// TIA Portal V20 export
DATA_BLOCK "MP101"   // DB181
// stored: MemoryReserve 100
   VAR
      "KISTLER 100KN PRESS POWER TRIPPED E202CB" : Bool;
      "KISTLER 100KN PRESS POWER TRIPPED E208CB" : Bool;
      "KISTLER 30KN PRESS POWER TRIPPED E214CB" : Bool;
      SPARE : Bool;
      SPARE_1 : Bool;
      "E8404PWS CONTROLLER POWER SMPS AC POWER TRIPPED E320CB" : Bool;
      "E8704PWS SAFETY POWER SMPS AC POWER TRIPPED E326CB" : Bool;
      "E8804PWS CONTRL POWER SMPS AC POWER TRIPPED E332CB" : Bool;
      "PROCESSOR POWER ON TIPPRED E4120CB" : Bool;
      "PROGRAMING POWER OUTLET TRPPED E4126CB" : Bool;
      SPARE_2 : Bool;
      "PANEL LED POWER TRIPPED E4304CB" : Bool;
      SPARE_3 : Bool;
      "PLC POWER SMPS DC OK E4404PWS" : Bool;
      "CONTROL LEVEL HUB POWER TRIPPED E4420CB" : Bool;
      "MAIN HMI POWER TRIPPED E4426CB" : Bool;
      "PORTABLE HMI POWER TIPPED E4432CB" : Bool;
      "PORTABLE HMI POWER TIPPED E4456CB" : Bool;
      "120VAC HEATER-1 POWER TR PRIMARY TRIPPED E5100CB" : Bool;
      SPARE_4 : Bool;
      SPARE_5 : Bool;
      "UPPER 1-1 HEATER POWER TRIPPED E5156CB" : Bool;
      "UPPER 1-2 HEATER POWER TRIPPED E5162CB" : Bool;
      "LOWER 1-1 HEATER POWER TRIPPED E5168CB" : Bool;
      "LOWER 1-2 HEATER POWER TRIPPED E5174CB" : Bool;
      "LOWER 1-3 HEATER POWER TRIPPED E5180CB" : Bool;
      SPARE_6 : Bool;
      "120VAC HEATER-2 POWER TR PRIMARY TRIPPED E6100CB" : Bool;
      SPARE_7 : Bool;
      SPARE_8 : Bool;
      "UPPER 2-1 HEATER POWER TRIPPED E6156CB" : Bool;
      "UPPER 2-2 HEATER POWER TRIPPED E6162CB" : Bool;
   END_VAR
BEGIN
END_DATA_BLOCK
